INTERFACE ITF_HMIEMenu EXTENDS ITF_BaseControlElement

METHOD PUBLIC GetNumberOfActriveScreen : INT
VAR_INPUT
END_VAR
END_METHOD

METHOD PUBLIC GetNumberOfAddedButton : INT
VAR_INPUT
END_VAR
END_METHOD

METHOD IsActiveButton : BOOL
VAR_INPUT
	iButton		: INT;	//numer przycisku
	bIN			: BOOL;
END_VAR
END_METHOD

METHOD PUBLIC IsChangePage : BOOL
VAR_INPUT
END_VAR
END_METHOD

METHOD IsEnableButton : BOOL
VAR_INPUT
	iButton		: INT;	//numer przycisku
	bIN			: BOOL;
END_VAR
END_METHOD

METHOD IsVisibleButton : BOOL
VAR_INPUT
	iButton		: INT;	//numer przycisku
	bIN			: BOOL;
END_VAR
END_METHOD

METHOD PUBLIC ResetChangePage
VAR_INPUT
END_VAR
END_METHOD

METHOD SetActiveButton : BOOL
VAR_INPUT
	iButton		: INT;	//numer przycisku
	bIN			: BOOL;
END_VAR
END_METHOD

METHOD SetEnableButton : BOOL
VAR_INPUT
	iButton		: INT;	//numer przycisku
	bIN			: BOOL;
END_VAR
END_METHOD

METHOD SetVisibleButton : BOOL
VAR_INPUT
	iButton		: INT;	//numer przycisku
	bIN			: BOOL;
END_VAR
END_METHOD

(*			
	RafalOS
	Rafał Osajda		11.11.2025		TC 4024.66
	testuje czy jest coś naciśnięte w menu i przełącza
*)
METHOD PUBLIC Testing : BOOL
END_METHOD

END_INTERFACE

(* stored: Version 1.1.0.1
   Itf ITF_HMIEMenu: Id {dc3b9d3c-c21c-4086-8483-fad3245993b2}
   Method GetNumberOfActriveScreen: Id {275bcb8b-dc1b-09bf-3fd0-fb5ccb6d63f4}
   Method GetNumberOfAddedButton: Id {cc008938-87b3-00fa-29a8-ecaf33db7187}
   Method IsActiveButton: Id {f22efdf8-7886-0a69-2875-61fb93444426}
   Method IsChangePage: Id {dcb8cd65-7abb-08aa-2f1f-e600eedf00fe}
   Method IsEnableButton: Id {72febfc2-fec1-00a8-30f0-9e1258ba32a6}
   Method IsVisibleButton: Id {c97994a9-d7c0-0cc8-398f-1e3c16523eda}
   Method ResetChangePage: Id {ce2966c9-f5be-0ebf-17d7-9b934a5a66ad}
   Method SetActiveButton: Id {32dcc8e6-c509-00e9-0dab-1d92581de236}
   Method SetEnableButton: Id {3c4c605a-1ecc-0462-26e5-8097143c9e41}
   Method SetVisibleButton: Id {748343ca-0118-07c9-326b-1ec360eba4bb}
   Method Testing: Id {83afaa7e-d27f-0216-156a-27abde1fe304} *)
